// TIA Portal V16 export
// export: Created 2021-05-25T16:14:41.4638669Z, ExportSetting WithDefaults, DisplayName Totally Integrated Automation Portal, DisplayVersion V16, DisplayName TIA Portal Version Control Interface, DisplayVersion V16, DisplayName TIA Portal Openness, DisplayVersion V16, DisplayName STEP 7 Professional, DisplayVersion V16, DisplayName STEP 7 Safety, DisplayVersion V16, DisplayName WinCC Unified SCADA Engineering System, DisplayVersion V16
DATA_BLOCK "dbPLCClock"   // DB251
{ S7_Optimized_Access := 'FALSE'; DB_Accessible_From_OPC_UA := 'FALSE' }
VERSION : 0.1
// stored: AutoNumber false, DBAccessibleFromOPCUA false, IsOnlyStoredInLoadMemory false, IsWriteProtectedInAS false
   VAR
      Tenth : Bool := FALSE;
      SEC : Bool := FALSE;
      Minute : Bool := FALSE;
      Hour : Bool := FALSE;
      Day : Bool := FALSE;
      Week : Bool := FALSE;
      Month : Bool := FALSE;
      Year : Bool := FALSE;
      SetPLCClock : Bool := FALSE;
      SetOPPLCClock : Bool := FALSE;
      PLC : "udtClock";
      SCADA : "udtClock";
      SweepTime : Int := 17;
      ScanCounter : Int := 72;
   END_VAR
BEGIN
END_DATA_BLOCK
